TYPE PLCStruct :
STRUCT
	inVal		AT %MD10: INT;
	floatVal	AT %MD14: REAL;
	boolVal		AT %MD18: BOOL;
END_STRUCT
END_TYPE

(* stored: Version 1.1.0.1, ProductVersion 3.1.4024.4
   DUT PLCStruct: Id {0dd5e1a9-15f9-45e3-9add-13db26208018} *)
